TYPE ST_QrScanMotionConfig :
STRUCT
    fVelocity : LREAL;
    fAcceleration : LREAL;
    fDeceleration : LREAL;
END_STRUCT
END_TYPE

(* stored: Version 1.1.0.1, ProductVersion 3.1.4026.20
   DUT ST_QrScanMotionConfig: Id {94d9524b-c253-48fa-8051-db3c2ea68776} *)
